FUNCTION_BLOCK GET_ANY (* Reads a ANY value from an InOut variable and provides it as a buffered Output *)
  (* Standard: 61499-1 *)
  (* Version 1.0, 2026-05-07, Gemini CLI, Initial version *)
  PACKAGE logiBUS::utils::conversion::provide;
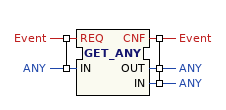
  EVENT_INPUT
    REQ WITH IN; (* Normal Execution Request *)
  END_EVENT
  EVENT_OUTPUT
    CNF WITH OUT, IN; (* Execution Confirmation *)
  END_EVENT
  VAR_OUTPUT
    OUT : ANY; (* Buffered output value *)
  END_VAR
  VAR_IN_OUT
    IN : ANY; (* Source variable (InOut) *)
  END_VAR
  EC_STATES
    REQ : REQ -> CNF;
  END_STATES
  ALGORITHM REQ IN ST: (* Read value from InOut source and store in local buffer *)
OUT := IN;
  END_ALGORITHM
END_FUNCTION_BLOCK
